{attribute 'reflection'}
FUNCTION_BLOCK FB_DebugMsg
(**************************************************************************************
 * 	Application		:	BoxControl Framework
 *	Revision		:	$Revision: 404529 $
 *	Revision date	:	$Date: 2018-04-23 08:21:38 +0200 (Mo., 23 Apr 2018) $
 *	Last changed by	:	$Author: b7bolm $
 *	URL				:	$URL: http://almscdc.swisslog.com/repo/SWPD/Development/BoxControlFramework/20_Release/trunk/01_Software/BCF/BCF/JumpStart/20_Product/10_App/11_Com/10_Lib/FB_DebugMsg.TcPOU $
 *
 *	Purpose			:	Debug massage
 *
 * ------------------------------------------------------------------------------------
 *	Copyright Swisslog [IP AG], Switzerland. All rights reserved.
 * 
 * ------------------------------------------------------------------------------------
 *	
 * 	Revision History: 
 *
 * VERSION DATE         INITIALS     DESCRIPTION
 * 0.0     DD.MM.YYYY   (name)       (explain customized modifications)
 *
 **************************************************************************************)
VAR
	{attribute 'instance-path'}
	{attribute 'no_init'}
	InstanceName				: STRING[System.DEBUGSOURCELENGTH];
	//------------------------------------------------------------------
	LastMessage					: STRING[System.DEBUGMESSAGELENGTH];
	fbGetCurTaskIdx				: GETCURTASKINDEX; // Returns the actual task index
	LastCycleCounterValue		: UDINT;
END_VAR

// Body never called

METHOD FB_init : BOOL

(********************************************************************************************************************************)
VAR_INPUT
	bInitRetains          : BOOL; // if TRUE, the retain variables are initialized (warm start / cold start)
	bInCopyCode           : BOOL;  // if TRUE, the instance afterwards gets moved into the copy code (online change)
  (*----------------------------------------------------------------------------------------------------------------------------*)
END_VAR

(********************************************************************************************************************************)
VAR
END_VAR

(********************************************************************************************************************************)
(** remove 'QB2Jumpstart.JumpStart.' from instance path *************************************************************************)
F_InstancePathRemovals(DestStart     := ADR(InstanceName),
                       DestEnd       := ADR(InstanceName) + SIZEOF(InstanceName),
                       RemoveLastPart:= TRUE);  




(********************************************************************************************************************************)
(** done ************************************************************************************************************************)
END_METHOD

METHOD M_SendErrorMsg
(**************************************************************************************
 * 	Application		:	BoxControl Framework
 *	Revision		:	$Revision: 404529 $
 *	Revision date	:	$Date: 2018-04-23 08:21:38 +0200 (Mo., 23 Apr 2018) $
 *	Last changed by	:	$Author: b7bolm $
 *	URL				:	$URL: http://almscdc.swisslog.com/repo/SWPD/Development/BoxControlFramework/20_Release/trunk/01_Software/BCF/BCF/JumpStart/20_Product/10_App/11_Com/10_Lib/FB_DebugMsg.TcPOU $
 *
 *	Purpose			:	Send error message
 *
 * ------------------------------------------------------------------------------------
 *	Copyright Swisslog [IP AG], Switzerland. All rights reserved.
 * 
 * ------------------------------------------------------------------------------------
 *	
 * 	Revision History: 
 *
 * 	VERSION			DATE			INITIALS			DESCRIPTION
 *	0.1				01.01.2001		swl					Example
 *
 **************************************************************************************)
VAR_INPUT
	mMessage	: STRING(System.DEBUGMESSAGELENGTH);
END_VAR
// message is not equal to last sent message
// same message can be sent in same cycle several times
fbDebugMsgManager.M_SendMessage(E_DebugMsgType.ERROR, InstanceName, ADR(mMessage), INT_TO_UDINT(LEN(mMessage)));
LastMessage := mMessage;
// Get current cycle count
fbGetCurTaskIdx();
LastCycleCounterValue := _TaskInfo[fbGetCurTaskIdx.index].CycleCount;
END_METHOD

METHOD M_SendInfoMsg
(**************************************************************************************
 * 	Application		:	BoxControl Framework
 *	Revision		:	$Revision: 404529 $
 *	Revision date	:	$Date: 2018-04-23 08:21:38 +0200 (Mo., 23 Apr 2018) $
 *	Last changed by	:	$Author: b7bolm $
 *	URL				:	$URL: http://almscdc.swisslog.com/repo/SWPD/Development/BoxControlFramework/20_Release/trunk/01_Software/BCF/BCF/JumpStart/20_Product/10_App/11_Com/10_Lib/FB_DebugMsg.TcPOU $
 *
 *	Purpose			:	Send info message
 *
 * ------------------------------------------------------------------------------------
 *	Copyright Swisslog [IP AG], Switzerland. All rights reserved.
 * 
 * ------------------------------------------------------------------------------------
 *	
 * 	Revision History: 
 *
 * 	VERSION			DATE			INITIALS			DESCRIPTION
 *	0.1				01.01.2001		swl					Example
 *
 **************************************************************************************)
VAR_INPUT
	mMessage			: STRING(System.DEBUGMESSAGELENGTH);
END_VAR
// message is not equal to last sent message
// same message can be sent in same cycle several times
fbDebugMsgManager.M_SendMessage(E_DebugMsgType.INFO, InstanceName, ADR(mMessage), INT_TO_UDINT(LEN(mMessage)));
LastMessage := mMessage;
// Get current cycle count
fbGetCurTaskIdx();
LastCycleCounterValue := _TaskInfo[fbGetCurTaskIdx.index].CycleCount;
END_METHOD

METHOD M_SendLongMsg
(**************************************************************************************
 * 	Application		:	BoxControl Framework
 *	Revision		:	$Revision: 404529 $
 *	Revision date	:	$Date: 2018-04-23 08:21:38 +0200 (Mo., 23 Apr 2018) $
 *	Last changed by	:	$Author: b7bolm $
 *	URL				:	$URL: http://almscdc.swisslog.com/repo/SWPD/Development/BoxControlFramework/20_Release/trunk/01_Software/BCF/BCF/JumpStart/20_Product/10_App/11_Com/10_Lib/FB_DebugMsg.TcPOU $
 *
 *	Purpose			:	Send long message
 *						Long messages will be separated in messages < MAX_STRING_LENGTH
 *						and forwarded as normal messages.
 *
 * ------------------------------------------------------------------------------------
 *	Copyright Swisslog [IP AG], Switzerland. All rights reserved.
 * 
 * ------------------------------------------------------------------------------------
 *	
 * 	Revision History: 
 *
 * 	VERSION			DATE			INITIALS			DESCRIPTION
 *	0.1				01.01.2001		swl					Example
 *
 **************************************************************************************)
VAR_INPUT
	mDebugMsgType	: E_DebugMsgType; // Message type
	mpData			: PVOID; // Address to data source
	mLen			: UDINT; // Length of the message (Attention, if the input is String use LEN instead of SIZEOF
END_VAR

// message is not equal to last sent message
// same message can be sent in same cycle several times
fbDebugMsgManager.M_SendMessage(mDebugMsgType, InstanceName, mpData, mLen);

// Store first 255 characters for debugging
F_BlockCopy(
	pSrc:= mpData, 
	LenSrc:= mLen, 
	pDest:= ADR(LastMessage), 
	LenDest:= SIZEOF(LastMessage));
	
// Get current cycle count
fbGetCurTaskIdx();
LastCycleCounterValue := _TaskInfo[fbGetCurTaskIdx.index].CycleCount;
END_METHOD

METHOD M_SendWarningMsg
(**************************************************************************************
 * 	Application		:	BoxControl Framework
 *	Revision		:	$Revision: 404529 $
 *	Revision date	:	$Date: 2018-04-23 08:21:38 +0200 (Mo., 23 Apr 2018) $
 *	Last changed by	:	$Author: b7bolm $
 *	URL				:	$URL: http://almscdc.swisslog.com/repo/SWPD/Development/BoxControlFramework/20_Release/trunk/01_Software/BCF/BCF/JumpStart/20_Product/10_App/11_Com/10_Lib/FB_DebugMsg.TcPOU $
 *
 *	Purpose			:	Send warning message
 *
 * ------------------------------------------------------------------------------------
 *	Copyright Swisslog [IP AG], Switzerland. All rights reserved.
 * 
 * ------------------------------------------------------------------------------------
 *	
 * 	Revision History: 
 *
 * 	VERSION			DATE			INITIALS			DESCRIPTION
 *	0.1				01.01.2001		swl					Example
 *
 **************************************************************************************)
VAR_INPUT
	mMessage		: STRING(System.DEBUGMESSAGELENGTH);
END_VAR
// message is not equal to last sent message
// same message can be sent in same cycle several times
fbDebugMsgManager.M_SendMessage(E_DebugMsgType.WARNING, InstanceName, ADR(mMessage), INT_TO_UDINT(LEN(mMessage)));
LastMessage := mMessage;
// Get current cycle count
fbGetCurTaskIdx();
LastCycleCounterValue := _TaskInfo[fbGetCurTaskIdx.index].CycleCount;;
END_METHOD

END_FUNCTION_BLOCK

(* stored: Version 1.1.0.1, ProductVersion 3.1.4024.4
   POU FB_DebugMsg: Id {9322272c-7c04-4b84-b82d-0944882a87ae}, SpecialFunc None
   Method FB_init: Id {4f740809-97e1-4bfe-b4e3-f490dcf8cf35}
   Method M_SendErrorMsg: Id {88cb378c-e8e9-4dda-a76b-f62e6b2d70cb}
   Method M_SendInfoMsg: Id {b25e85b6-2c1f-459b-8c0c-98cb0a02ee42}
   Method M_SendLongMsg: Id {b4441626-6749-46b6-86d1-1c75db5e54a9}
   Method M_SendWarningMsg: Id {565269e8-1618-4732-85f8-fc3b1deaba55} *)
